# EPICS autosave request: iocBoot/iocUSB1608G/auto_settings.req
file "1608G_settings.req", P=1608G:
